INTERFACE IList EXTENDS IReadOnlyList

METHOD Append : DINT
VAR_INPUT
	value : ANY;
	isObject : BOOL := FALSE;
END_VAR
END_METHOD

METHOD Clear
END_METHOD

METHOD Insert
VAR_INPUT
	value : ANY;
	index : DINT;
	isObject : BOOL := FALSE;
END_VAR
END_METHOD

METHOD RemoveAt
VAR_INPUT
	index : DINT;
END_VAR
END_METHOD

METHOD RemoveFirst : BOOL
VAR_INPUT
	value : ANY;
	isObject : BOOL := FALSE;
END_VAR
END_METHOD

METHOD RemoveMatched : DINT
VAR_INPUT
	predicate : IPredicate;
	skip : UDINT := 0;
	maxRemoved : UDINT := 16#FFFFFFFF;
END_VAR
END_METHOD

METHOD Set
VAR_INPUT
	value : ANY;
	index : DINT;
	isObject : BOOL := FALSE;
END_VAR
END_METHOD

END_INTERFACE

(* stored: Version 1.1.0.1
   Itf IList: Id {9c3b1d1d-e3a1-4bce-bd52-5e0052f367c5}
   Method Append: Id {ac3e836f-588d-4e01-b78d-500901973fe6}
   Method Clear: Id {ba38f8c3-7bfc-4319-b27d-1f0e4f4a811e}
   Method Insert: Id {5cb4df9f-a6c0-45ea-9622-2c963ebd948e}
   Method RemoveAt: Id {0b8aa929-5f9c-41a5-aea3-f997d9db63e1}
   Method RemoveFirst: Id {aef0ca9c-d714-4a50-863d-5b01a18245b0}
   Method RemoveMatched: Id {a4ece42e-52ea-4d71-9b54-b1ead6bc0e27}
   Method Set: Id {dd495513-6def-416e-84d8-dbee11dfb071} *)
